TYPE TrayLoad_IO_typ:
STRUCT
	Inputs	: TrayLoad_Inputs_typ;
	Outputs	: TrayLoad_Outputs_typ;
END_STRUCT
END_TYPE

(* stored: Version 1.1.0.1, ProductVersion 3.1.4024.12
   DUT TrayLoad_IO_typ: Id {ea677e51-681c-06ee-2706-9e6e36ab5c0f} *)
